(* Logix 5000 project; controller Lab8_3 5069-L306ERM rev 35.11; software revision 35.03 *)

TASK MainTask (continuous, watchdog 500 ms) : Lab8_3

MODULES
   Local : 5069-L306ERM (5069 0, rev 35.11)
      IOHub : vendor 1 type 7 code 358 (Ethernet 192.168.105.5, rev 1.1, Output RPI 20 ms)
END_MODULES

PROGRAM Lab8_3   (* main routine Lab8_3 *)
VAR
   MyTime : DINT[6];
   time : DINT;
END_VAR

ROUTINE Lab8_3   (* structured text *)
   
END_ROUTINE

ROUTINE random   (* structured text *)
   GSV(WallClockTime, , LocalDateTime, MyTime[0]);
   // Output:= [(MyTime[0]) mod (max - min + 1) ] + min
   
   
END_ROUTINE
END_PROGRAM
